Universal Robots PolyScope program: fun1.urp

Program fun1 (installation=default directory=/programs createdIn=5.9.1.1031110 lastSavedIn=5.9.1.1031110 robotSerialNumber=20195501059)
Calibrated DH parameters: a=[0.000146, -0.418764, -0.053981, 0.000058, -0.000023, 0]; d=[0.162545, 37.319448, -206.067439, 168.881546, 0.09955, 0.099464]; alpha=[1.57004, -0.001979, 0.002304, 1.570607, -1.57066, 0]; deltaTheta=[0, -0.174616, -1.258233, 1.432844, -0.000001, 0]
Robot Program (runOnlyOnce=true)
  URCap Gripper Activate (Robotiq_Grippers, Robotiq Inc.) dataModel(ResetAndActivateKey=false)
  URCap Gripper (Robotiq_Grippers, Robotiq Inc.) dataModel(position=100.0, force=100.0, speed=100.0, positionInDouble=100.0, forceInDouble=100.0, speedInDouble=100.0, slaveIds=[9], blocking=true)
  MoveJ speed 60 deg/s, acceleration 80 deg/s^2 (useActiveTCP=true) feature=Base
    Waypoint Waypoint_1: TCP in base x=107.132 y=-470.476 z=45.783 mm, rx=-2.748 ry=-1.5224 rz=-0.0001 rad; joints [86.737, -80.237, 122.137, -131.891, 270.059, -241.197] deg; TCP offset x=0 y=0 z=174 mm, rx=0 ry=0 rz=0 rad
  MoveL speed 250 mm/s, acceleration 1200 mm/s^2 (useActiveTCP=true) feature=Base
    Waypoint Waypoint_2: TCP in base x=312.793 y=-375.091 z=64.537 mm, rx=2.7481 ry=1.5224 rz=0 rad; joints [113.934, -81.41, 119.992, -128.575, 270.057, -214.004] deg
  URCap Olis Teleop (Olis Teleop, Olis Robotics)
  MoveL speed 250 mm/s, acceleration 1200 mm/s^2 (useActiveTCP=true) feature=Base
    Waypoint Waypoint_1: TCP in base x=107.132 y=-470.476 z=45.783 mm, rx=-2.748 ry=-1.5224 rz=-0.0001 rad; joints [86.737, -80.237, 122.137, -131.891, 270.059, -241.197] deg
